PROGRAM prgLab05_07
VAR
	i: INT;
END_VAR

//Na segunda parte desse mesmo exercício o objetivo é basicamente de expandí-lo transformando o que era um único
//Elemento em um vetor de 3

FOR i:=1 TO 3 DO
	IF GVL.aRooms[i].OccupancySensor THEN
		GVL.aRooms[i].Lighting:=TRUE;
		IF GVL.aRooms[i].Temp > 24 THEN
			GVL.aRooms[i].Heating:=FALSE;
		ELSIF GVL.aRooms[i].Temp <20 THEN
			GVL.aRooms[i].Heating:=TRUE;	
		END_IF
	ELSE
		GVL.aRooms[i].Lighting:=GVL.aRooms[i].Heating:=FALSE;	
	END_IF
	IF GVL.aRooms[i].AirQuality >= GVL.aRooms[i].setpoint THEN
		GVL.aRooms[i].Ventilation:=TRUE;
	ELSE
		GVL.aRooms[i].Ventilation:=FALSE;	
	END_IF	
	//Solução Lab 07
	IF GVL.aRooms[i].Temp< 20 THEN
		GVL.aRooms[i].status:= E_ROOM_TEMP_STS.baixa;
	ELSIF GVL.aRooms[i].Temp >=20 AND GVL.aRooms[i].Temp < 24 THEN
		GVL.aRooms[i].status:= E_ROOM_TEMP_STS.normal;
	ELSIF GVL.aRooms[i].Temp >=24 AND GVL.aRooms[i].Temp < 27 THEN
		GVL.aRooms[i].status:= E_ROOM_TEMP_STS.moderada;
	ELSIF GVL.aRooms[i].Temp >=27 AND GVL.aRooms[i].Temp < 32 THEN
		GVL.aRooms[i].status:= E_ROOM_TEMP_STS.alta;
	ELSIF GVL.aRooms[i].Temp >=32 THEN
		GVL.aRooms[i].status:= E_ROOM_TEMP_STS.muito_alta;
	END_IF	
END_FOR

END_PROGRAM

(* stored: Version 1.1.0.1, ProductVersion 3.1.4024.11
   POU prgLab05_07: Id {00ba17da-63d6-4e5f-a89a-1f7c6ef8a3c2}, SpecialFunc None *)
